{attribute 'GeneratedUsingTerminal: EL6851-0010-0016'}
{attribute addProperty BoxType "EL6851-0010-0016"}
{attribute addProperty Id "Receive_toggleAT %I*BOOL1Framing_errorAT %I*BOOL1Overrun_errorAT %I*BOOL1TxPDO_StateAT %I*BOOL1TxPDO_ToggleAT %I*BOOL1Channel_lengthAT %I*UINT2Start_codeAT %I*USINT1"}
{attribute addProperty CRC "1590553278"}
{attribute addProperty Size "8"}
TYPE DMX_Status_5ECDEABE :
STRUCT
	{attribute addProperty Name "Receive_toggle"}
	Receive_toggle AT %I* : BOOL;
	{attribute addProperty Name "Framing_error"}
	Framing_error AT %I* : BOOL;
	{attribute addProperty Name "Overrun_error"}
	Overrun_error AT %I* : BOOL;
	{attribute addProperty Name "TxPDO_State"}
	TxPDO_State AT %I* : BOOL;
	{attribute addProperty Name "TxPDO_Toggle"}
	TxPDO_Toggle AT %I* : BOOL;
	{attribute addProperty Name "Channel_length"}
	Channel_length AT %I* : UINT;
	{attribute addProperty Name "Start_code"}
	Start_code AT %I* : USINT;
END_STRUCT
END_TYPE

(* stored: Version 1.2.0.0, ProductVersion 3.1.4024.9
   DUT DMX_Status_5ECDEABE: Id {38e15b7c-fa9d-47c1-8a41-42e7c11ced3a} *)
